// TIA Portal V19 export
ORGANIZATION_BLOCK "MC_PreInterpolator"   // OB68, LAD, PreInterpolator
// stored: IsIECCheckEnabled true, SetENOAutomatically true
   VAR_INPUT
      Initial_Call : Bool;
      PIP_Input : Bool;
      PIP_Output : Bool;
      IO_System : USInt;
      Event_Count : Int;
      Reduction : UInt;
      CycleTime : UDInt;
   END_VAR
BEGIN

REGION Network 1: Call FB CalledInPreInterpolator from EM2
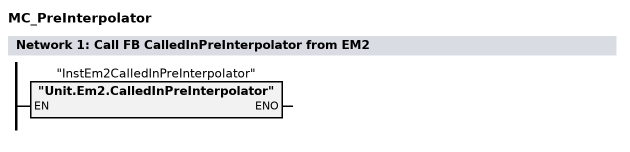
   RUNG wire#powerrail
      "InstEm2CalledInPreInterpolator"()
   END_RUNG
   // the same network as SCL:
   "InstEm2CalledInPreInterpolator"();   // "Unit.Em2.CalledInPreInterpolator"
END_REGION
END_ORGANIZATION_BLOCK
